FUNCTION_BLOCK EmergencyReactor_2 (* CAT Function Block Type *)
  (* Standard: 61499-2 *)
  (* Version 0.0, 7/4/2026, Schneider Electric, template *)
  PACKAGE SE.Nereda;
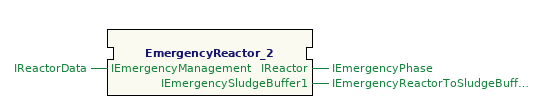
  SOCKETS
    IEmergencyManagement : IReactorData;
  END_SOCKETS
  PLUGS
    IReactor : IEmergencyPhase;
    IEmergencySludgeBuffer1 : IEmergencyReactorToSludgeBuffer;
  END_PLUGS
  (* 01 - FUNCTIONNAL INPUT INTERFACE *)
  (* 00 - INITIALIZATION *)
  (* 05 - LOGIC *)
  (* 06 - HMI INTERFACE *)
  (* 03 - FIELD INTERFACE *)
  (* 02 - FUNCTIONNAL OUTPUT INTERFACE *)
  (* Emergency Recipe Logic *)
  (* 04 - CHILDREN *)
  (* 4A - TYPICALS *)
  (* Reset Force Trs *)
  (* Skip Sludge Discharge Logic *)
  (* Steps Durations *)
  FBS
    INIT : plcStart(Prio := 50, Delay := T#0ms);
    IThis : EmergencyReactor_2_HMI(QI := TRUE);
    Step1_Feed : E_DELAY_V_D_ZERO;
    Step2_VentSludge : E_DELAY_V_D_ZERO;
    Step3_SludgeDischarge : E_DELAY_V_D_ZERO;
    Step4_LowerLevel : E_DELAY_V_D_ZERO;
    Step6_VentAerate : E_DELAY_V_D_ZERO;
    Step7_Wait : E_DELAY_V_D_ZERO;
    Step8_VentSludge : E_DELAY_V_D_ZERO;
    ResetTrsDelay : E_DELAY(DT := T#300ms);
    ResetTrs : TriggerNot0; {SET_ATTRIBUTE(Configuration.Component.HideUnusedPorts, )}
    SkipSludgeDischargeLogic : S1SkipS2(pin_EE0DFC875BC8FD2C := 3, pin_8745D113BFC82E09 := 9);
    SmoothSkip : boolValueChanged;
    EmergencyInitialisation : EmergencyInit2(pin_F6BF5230E0E343F0 := T#15m);
    S5_AerateTime : S5_AerateTime2;
    Step5_Aerate : COUNTER(pin_12B31DD3EC852BD8 := TRUE); {SET_ATTRIBUTE(Configuration.Component.HideUnusedPorts, )}
    ForceStopAeration : StopAerate2;
    FeedStarted : boolValueChanged;
    GoToS8 : OR_88A3DD8EC65DD11C; {SET_ATTRIBUTE(Configuration.GenericFBType.InterfaceParams, Runtime.Standard#CNT:=2;OUT:BOOL)}
    GoToS8Smooth : boolValueChanged;
    EmergencyRecipeSequence : EmergencyRecipeSequence_2;
    Step9_SludgeDischarge : E_DELAY_V_D_ZERO;
    Step10_Wait : E_DELAY_V_D_ZERO;
    Step6_VentAerate1 : E_DELAY_V_D_ZERO;
  END_FBS
  EVENT_CONNECTIONS
    IReactor.3CBA18632C5993F7 TO EmergencyRecipeSequence.5F230DB7635D55AE;
    IReactor.B9A3DD1A626C862D TO EmergencyRecipeSequence.5F230DB7635D55AE;
    IReactor.4DCB92F6993C5EE1 TO EmergencyRecipeSequence.5F230DB7635D55AE;
    IReactor.CF95EBECB4A2EBBE TO EmergencyRecipeSequence.5F230DB7635D55AE;
    IReactor.3F1D0A688A5176FD TO EmergencyRecipeSequence.5F230DB7635D55AE;
    IReactor.B334EFD88038E789 TO EmergencyRecipeSequence.5F230DB7635D55AE;
    Step1_Feed.1457E63E0C241C83 TO EmergencyRecipeSequence.62A0C79B5D89C4FB;
    Step2_VentSludge.1457E63E0C241C83 TO EmergencyRecipeSequence.24741A0901B103DB;
    Step3_SludgeDischarge.1457E63E0C241C83 TO EmergencyRecipeSequence.FEA4481ED0C2A43C;
    Step4_LowerLevel.1457E63E0C241C83 TO EmergencyRecipeSequence.9041C273A86FC2E4;
    Step6_VentAerate.1457E63E0C241C83 TO EmergencyRecipeSequence.5D1CA06DD981DC88;
    Step7_Wait.1457E63E0C241C83 TO EmergencyRecipeSequence.87133753EE03EF50;
    Step8_VentSludge.1457E63E0C241C83 TO EmergencyRecipeSequence.45085FB160311A79;
    SmoothSkip.CHD TO EmergencyRecipeSequence.3824F5F239920D6C;
    IReactor.1F4F3B9CDE5DCB1C TO EmergencyRecipeSequence.F6AE117EB4EE709F;
    IReactor.0001D958FDF5E959 TO EmergencyRecipeSequence.C960811A6435E9DC;
    EmergencyRecipeSequence.3B7FC9F46DCC7431 TO IReactor.42529785B6820948;
    EmergencyRecipeSequence.3B7FC9F46DCC7431 TO IReactor.B633B7A44F850807;
    EmergencyRecipeSequence.3B7FC9F46DCC7431 TO IReactor.B3BCF5E9C62C69B8;
    EmergencyRecipeSequence.3B7FC9F46DCC7431 TO IReactor.2000F66036015D52;
    EmergencyRecipeSequence.3B7FC9F46DCC7431 TO IReactor.8A3A142CC73C9F25;
    EmergencyRecipeSequence.BFFB06EAE80CA24C TO Step1_Feed.START;
    EmergencyRecipeSequence.899C844BE45E6C4D TO Step1_Feed.STOP;
    EmergencyRecipeSequence.758107C20AA8F48B TO Step2_VentSludge.START;
    EmergencyRecipeSequence.18CD3557BE39D07B TO Step2_VentSludge.STOP;
    EmergencyRecipeSequence.77F2040F9E65C9AB TO Step3_SludgeDischarge.START;
    EmergencyRecipeSequence.728874E1FE8923C2 TO Step3_SludgeDischarge.STOP;
    EmergencyRecipeSequence.F0D24A0013391FCB TO Step4_LowerLevel.START;
    EmergencyRecipeSequence.DBC21B10FAB6B6D6 TO Step4_LowerLevel.STOP;
    EmergencyRecipeSequence.5F688AB98BE3DBA8 TO Step5_Aerate.START;
    EmergencyRecipeSequence.CFC9FFB1D070A85D TO Step5_Aerate.STOP;
    EmergencyRecipeSequence.D93FC42377801178 TO Step6_VentAerate.START;
    EmergencyRecipeSequence.94B7CB1BE3844802 TO Step6_VentAerate.STOP;
    EmergencyRecipeSequence.D6AAA325013931BD TO Step7_Wait.START;
    EmergencyRecipeSequence.66DEB21CDAAC07A1 TO Step7_Wait.STOP;
    EmergencyRecipeSequence.4C7C51E8F73DAAF0 TO Step8_VentSludge.START;
    EmergencyRecipeSequence.4F8F2BAA25498729 TO Step8_VentSludge.STOP;
    Step1_Feed.INITO TO Step2_VentSludge.INIT;
    Step2_VentSludge.INITO TO Step3_SludgeDischarge.INIT;
    Step3_SludgeDischarge.INITO TO Step4_LowerLevel.INIT;
    Step4_LowerLevel.INITO TO Step6_VentAerate1.INIT;
    Step6_VentAerate.INITO TO Step7_Wait.INIT;
    Step7_Wait.INITO TO Step8_VentSludge.INIT;
    ResetTrs.4D14044435EE07B0 TO ResetTrsDelay.START;
    SkipSludgeDischargeLogic.9D8BC655F08DCD6C TO SmoothSkip.REQ;
    EmergencyRecipeSequence.556D2F5B235B9790 TO SkipSludgeDischargeLogic.74AB0FAFF377F024;
    IEmergencyManagement.E1D373823D64ACA0 TO IReactor.0FA2667D36826F2B;
    Step5_Aerate.INITO TO EmergencyInitialisation.7772EF333A96DB94;
    EmergencyInitialisation.5BE6234FD14189DB TO INIT.ACK_FIRST;
    EmergencyInitialisation.87FEA01C25C77B1D TO EmergencyRecipeSequence.4E3261F33DF95CD1;
    IEmergencyManagement.9D1E5F7369C5538B TO EmergencyInitialisation.E815AC1CDB9AD32A;
    IEmergencyManagement.E1D373823D64ACA0 TO EmergencyInitialisation.1FA17325B39B02F6;
    IEmergencyManagement.61CD32E3E6AEDF7D TO EmergencyInitialisation.5DED6604D26A7975;
    IEmergencyManagement.198EF041C70827BC TO S5_AerateTime.0D2EA60FD6C23367;
    IEmergencyManagement.1C1DD8946F24CFF9 TO S5_AerateTime.C7A276F0816E041D;
    S5_AerateTime.8B394E005AFEAD78 TO IEmergencyManagement.D499D06F1953A020;
    S5_AerateTime.8B394E005AFEAD78 TO Step5_Aerate.E9D3BB8F75D35902;
    IEmergencyManagement.7D5F3067068DE334 TO EmergencyRecipeSequence.25F0D728C2D36669;
    IEmergencyManagement.7D5F3067068DE334 TO IReactor.3CAF22C03BECB249;
    ForceStopAeration.7530111629E0F796 TO EmergencyRecipeSequence.56BBB9AD7704F212;
    IReactor.B9A3DD1A626C862D TO ForceStopAeration.D950482A44AC5C73;
    IEmergencyManagement.B3BDDBF095B97A2B TO ForceStopAeration.D950482A44AC5C73;
    IEmergencyManagement.E1D373823D64ACA0 TO EmergencyRecipeSequence.68E2F3B4BFF358D6;
    IReactor.3CBA18632C5993F7 TO FeedStarted.REQ;
    FeedStarted.CHD TO IEmergencyManagement.138EEC247A2C05E7;
    SkipSludgeDischargeLogic.5213FB99EC5BE951 TO ForceStopAeration.D950482A44AC5C73;
    EmergencyInitialisation.5BE6234FD14189DB TO EmergencyRecipeSequence.68E2F3B4BFF358D6;
    IEmergencyManagement.395F2A7D1AB6A478 TO EmergencyInitialisation.8D22CD40FC41E8B5;
    IEmergencyManagement.395F2A7D1AB6A478 TO EmergencyRecipeSequence.8BD9ED85505D599F;
    Step6_VentAerate1.INITO TO Step6_VentAerate.INIT;
    IEmergencyManagement.CF316F4BA7C11A07 TO EmergencyInitialisation.2B59ADD28234FD73;
    IEmergencyManagement.77175193A5DFB16A TO EmergencyRecipeSequence.CF595DA908C4D604;
    EmergencyRecipeSequence.556D2F5B235B9790 TO IEmergencyManagement.48081868B719DABE;
    IReactor.4DCB92F6993C5EE1 TO IEmergencyManagement.48081868B719DABE;
    GoToS8.CNF TO GoToS8Smooth.REQ;
    GoToS8Smooth.CHD TO EmergencyRecipeSequence.4E3261F33DF95CD1;
    EmergencyInitialisation.87FEA01C25C77B1D TO GoToS8.REQ;
    IEmergencyManagement.61CD32E3E6AEDF7D TO GoToS8.REQ;
    Step9_SludgeDischarge.INITO TO Step10_Wait.INIT;
    Step8_VentSludge.INITO TO Step9_SludgeDischarge.INIT;
    EmergencyRecipeSequence.159DAAF64474114A TO Step9_SludgeDischarge.START;
    EmergencyRecipeSequence.043FC99FF466ACE5 TO Step9_SludgeDischarge.STOP;
    EmergencyRecipeSequence.6D74F5F87D5293B0 TO Step10_Wait.START;
    EmergencyRecipeSequence.C125C1F9A17D8460 TO Step10_Wait.STOP;
    Step9_SludgeDischarge.1457E63E0C241C83 TO EmergencyRecipeSequence.CBB132F8E1E06425;
    Step10_Wait.1457E63E0C241C83 TO EmergencyRecipeSequence.2C1A1FFEA773D0E8;
    EmergencyRecipeSequence.3B7FC9F46DCC7431 TO IReactor.0F544A40694CE400;
    EmergencyRecipeSequence.556D2F5B235B9790 TO IReactor.DAE1720DE74FAACB;
    IEmergencyManagement.93812D9FEC4294F9 TO EmergencyRecipeSequence.035DD9202D5272B8;
    Step10_Wait.INITO TO Step5_Aerate.INIT;
    EmergencyRecipeSequence.5F688AB98BE3DBA8 TO Step6_VentAerate1.START;
    EmergencyRecipeSequence.CFC9FFB1D070A85D TO Step6_VentAerate1.STOP;
    Step6_VentAerate1.1457E63E0C241C83 TO EmergencyRecipeSequence.AA8C7EBD4EBD70F0;
    IReactor.2DDA8AB533D7441D TO EmergencyRecipeSequence.1E0B2A3AB6A90076;
    IEmergencyManagement.E1D373823D64ACA0 TO IEmergencySludgeBuffer1.D46CB75BB047204F;
    IReactor.3CBA18632C5993F7 TO IEmergencySludgeBuffer1.3F9F1A3D0BC5ACBF;
    IEmergencyManagement.7D5F3067068DE334 TO IEmergencySludgeBuffer1.69A30D6F1EEC778E;
    INIT.FIRST_INIT TO IThis.11B0EEC0AF1F6F5A;
    INIT.REDO_INIT TO IThis.11B0EEC0AF1F6F5A;
    EmergencyRecipeSequence.556D2F5B235B9790 TO IThis.C39B00E2AD0232CC;
    IEmergencyManagement.E1D373823D64ACA0 TO IThis.C454C4B6A808EB9F;
    ResetTrsDelay.EO TO IThis.908B60AA8FD99187;
    IThis.7797C5138BE465AE TO IThis.D73F4F826029EE6B;
    S5_AerateTime.8B394E005AFEAD78 TO IThis.188CF7222009AE29;
    ForceStopAeration.5ED5F3C70645AC06 TO IThis.188CF7222009AE29;
    S5_AerateTime.878A4998A65F56E0 TO IThis.7360449561F94EA9;
    Step5_Aerate.INITO TO IThis.9D2FDC03CB586F4F;
    IEmergencyManagement.7D5F3067068DE334 TO IThis.FD84EE6824F2A446;
    IThis.69E91E9E46EEE4A5 TO Step1_Feed.INIT;
    IThis.7C2D7DF8D7E29126 TO ResetTrs.98B4D14610C64DF9;
    IThis.7C2D7DF8D7E29126 TO EmergencyRecipeSequence.56F42E6AA601D269;
    IThis.A02D1390759D9486 TO EmergencyInitialisation.4A8FE6F9318E2B02;
    IThis.A02D1390759D9486 TO S5_AerateTime.0D2EA60FD6C23367;
    IThis.A02D1390759D9486 TO ForceStopAeration.D950482A44AC5C73;
    IThis.1D92FE3FE5B995E2 TO IReactor.BC34E8F0E0F52444;
    IThis.621A8557BCE5A33F TO IReactor.1BDE0720AC8B4391;
    IThis.72CBF4E7BB40B16D TO IReactor.FF8E2C9D67AADBF4;
    IThis.024A635046F06C0B TO IReactor.4E395DC016F294D9;
  END_CONNECTIONS
  DATA_CONNECTIONS
    EmergencyRecipeSequence.8B42F21C51560908 TO IReactor.8B7B31E6EA54014D;
    EmergencyRecipeSequence.A11B93FCF2C8455F TO IReactor.09084E8C7BADBD46;
    EmergencyRecipeSequence.2A15B42D80F87BCA TO IReactor.C947D1396F3B0873;
    EmergencyRecipeSequence.EC54CA5500C858C1 TO IReactor.419E697BA1D2FB08;
    EmergencyRecipeSequence.A9E8FE003DEE6E89 TO IReactor.C584AEAB998AB515;
    IReactor.599667ECF678E518 TO EmergencyRecipeSequence.02C5FE17473E63ED;
    IReactor.656FC0E59D395E4C TO EmergencyRecipeSequence.9F29B8C1612DCC07;
    IReactor.9CFBB312DE29B9C4 TO EmergencyRecipeSequence.ED57F4FA4B77207F;
    IReactor.A1460632301E8B7F TO EmergencyRecipeSequence.89F466D1EDD34A8F;
    IReactor.A92252B4F4DF917A TO EmergencyRecipeSequence.5FBA38ABF9198C98;
    Step1_Feed.716D3F3042596C89 TO EmergencyRecipeSequence.CA116731A496187E;
    Step2_VentSludge.716D3F3042596C89 TO EmergencyRecipeSequence.356882B50FEB9A7D;
    Step3_SludgeDischarge.716D3F3042596C89 TO EmergencyRecipeSequence.111361C8BEDF440B;
    Step4_LowerLevel.716D3F3042596C89 TO EmergencyRecipeSequence.82CEB92F735FC5D4;
    Step6_VentAerate.716D3F3042596C89 TO EmergencyRecipeSequence.0228D93DF2A0E691;
    Step7_Wait.716D3F3042596C89 TO EmergencyRecipeSequence.F00C171ABB730806;
    Step8_VentSludge.716D3F3042596C89 TO EmergencyRecipeSequence.0EEA3AF033FFC1FD;
    SmoothSkip.Output TO EmergencyRecipeSequence.43A591812296CA90;
    IReactor.579DEB3758BDB938 TO EmergencyRecipeSequence.7A1CAB8AE52AE374;
    IReactor.1156E288C0C38120 TO EmergencyRecipeSequence.CB5D14E9C5586FB9;
    SkipSludgeDischargeLogic.DBD9C05F71A70F66 TO SmoothSkip.Input;
    EmergencyRecipeSequence.1A64065878672AC0 TO SkipSludgeDischargeLogic.2058267BFC81675C;
    IEmergencyManagement.F0BEEA13B7FB6780 TO IReactor.5159724764416574;
    EmergencyInitialisation.AC3533DBCBFC24D5 TO EmergencyRecipeSequence.73A0EB798F8AE64D;
    GoToS8Smooth.Output TO EmergencyRecipeSequence.8C498327642AF905;
    IEmergencyManagement.7614E537E01F969F TO EmergencyInitialisation.C2EDD382E854309C;
    IEmergencyManagement.852A82A24B95110C TO EmergencyInitialisation.8DFF8A8B75E55DBC;
    IEmergencyManagement.F0BEEA13B7FB6780 TO EmergencyInitialisation.5CEC0909DD41DD44;
    IEmergencyManagement.074948F0B024FF2E TO EmergencyInitialisation.417A4B99C6EAD037;
    IEmergencyManagement.758E7E3A994DF6A3 TO S5_AerateTime.051E4CDC84405E95;
    IEmergencyManagement.90388C221FF11A3D TO S5_AerateTime.4E488DE24686A5F2;
    S5_AerateTime.3E8F4A267A25DD05 TO IEmergencyManagement.793E1D04BE895F4E;
    S5_AerateTime.6A9E00F95DC3CAB2 TO IEmergencyManagement.3807C75A82F33B22;
    S5_AerateTime.3E8F4A267A25DD05 TO Step5_Aerate.2BD9889911508ED1;
    IEmergencyManagement.35F3027F47B7A966 TO EmergencyRecipeSequence.53ADC5A2738A60DC;
    IEmergencyManagement.35F3027F47B7A966 TO IReactor.63583CB69DED3592;
    ForceStopAeration.8A55773E02AECBCB TO EmergencyRecipeSequence.F39141D7A6A53184;
    IReactor.A63167A113600EB8 TO ForceStopAeration.19D48581CC6CEC95;
    IEmergencyManagement.83DE9B371B83EBB9 TO ForceStopAeration.20B8DEE9B9067A7E;
    IEmergencyManagement.F0BEEA13B7FB6780 TO EmergencyRecipeSequence.C537A25E1616B854;
    IReactor.F208B10244BCFEF2 TO FeedStarted.Input;
    FeedStarted.Output TO IEmergencyManagement.1D99A7E687AA4E06;
    IEmergencyManagement.3C27B3AC98B413B4 TO EmergencyInitialisation.79C2DD791585EF12;
    SkipSludgeDischargeLogic.59D0E2CFD06FCCA4 TO ForceStopAeration.E5E5D63C44355F3C;
    SkipSludgeDischargeLogic.BEF2F356EA04F63C TO ForceStopAeration.11917BAB3534074F;
    IEmergencyManagement.B1FC30AB336AE8E9 TO EmergencyRecipeSequence.EB24B639967D6395;
    EmergencyInitialisation.511C6D20E2A2A314 TO EmergencyRecipeSequence.A0CAD84FAFB4D508;
    IEmergencyManagement.B1FC30AB336AE8E9 TO EmergencyInitialisation.0058582DF67974BB;
    IEmergencyManagement.7FC77B7D4B4A5A4D TO EmergencyInitialisation.E3C04CDD1BC5A85D;
    IEmergencyManagement.B7D7393A43236C58 TO EmergencyInitialisation.9E91693CC077CF71;
    IEmergencyManagement.EEDAEC65A069032E TO EmergencyRecipeSequence.DB0738E6DF6AD68E;
    EmergencyRecipeSequence.1A64065878672AC0 TO IEmergencyManagement.613E286D19768818;
    IReactor.9CFBB312DE29B9C4 TO IEmergencyManagement.B3BCA5E1F4B3D013;
    GoToS8.OUT TO GoToS8Smooth.Input;
    EmergencyInitialisation.DF25ED8EB3FED3D4 TO GoToS8.IN1;
    IEmergencyManagement.713BAA92BE7C280E TO GoToS8.IN2;
    EmergencyRecipeSequence.05803EDF26892491 TO IReactor.198FB8D9804ED082;
    EmergencyRecipeSequence.4076D29063AB0B00 TO IReactor.486306180C62B9EF;
    IReactor.E996774D431E1B79 TO EmergencyRecipeSequence.A2ED29C3A4B57D44;
    IReactor.800D089965342DF6 TO EmergencyRecipeSequence.69F1D0FE13048380;
    Step9_SludgeDischarge.716D3F3042596C89 TO EmergencyRecipeSequence.CC3E20D91936F86E;
    Step10_Wait.716D3F3042596C89 TO EmergencyRecipeSequence.34AB02FCEF6642EF;
    IEmergencyManagement.1675BB23EEFCF5E9 TO EmergencyRecipeSequence.5989C017FA1C720B;
    Step6_VentAerate1.716D3F3042596C89 TO EmergencyRecipeSequence.CC0CCEB2D046659B;
    IReactor.C54C3886CAD71D0C TO EmergencyRecipeSequence.ACB986D17AA81EAF;
    IEmergencyManagement.F0BEEA13B7FB6780 TO IEmergencySludgeBuffer1.128C534CB06CDD0F;
    IReactor.D62F1904A2304A82 TO IEmergencySludgeBuffer1.D455BE5F3243F8CD;
    IReactor.EDD981DC30DF57BC TO IEmergencySludgeBuffer1.98FFA78276DA0653;
    IReactor.DA119668EC2B3E62 TO IEmergencySludgeBuffer1.2680CB24DDCC2D3E;
    IEmergencyManagement.35F3027F47B7A966 TO IEmergencySludgeBuffer1.A351B45A56D7A52F;
    EmergencyRecipeSequence.1A64065878672AC0 TO IThis.B3535F417A0074C5;
    IEmergencyManagement.F0BEEA13B7FB6780 TO IThis.71DB4288F980DD7A;
    IThis.F0EDDD752FB146AF TO IThis.2A6B48A49CC51EE0;
    S5_AerateTime.3E8F4A267A25DD05 TO IThis.0DCF6DA005733527;
    ForceStopAeration.C8B85A94FE68EF0C TO IThis.71E3BF00CD92D001;
    S5_AerateTime.4CD884F27F8D62DD TO IThis.A4518E9C005FED53;
    IEmergencyManagement.35F3027F47B7A966 TO IThis.7498551BC2E13233;
    IThis.5C9558FA20CCCAFB TO ResetTrs.622EA78CA147C620;
    IThis.5C9558FA20CCCAFB TO EmergencyRecipeSequence.1EFAFB1416CAAE87;
    IThis.D3644ED70524C0F1 TO Step1_Feed.DT1;
    IThis.D3644ED70524C0F1 TO S5_AerateTime.C5F8AE19B1F00F21;
    IThis.33D4356E329ECCF2 TO Step2_VentSludge.DT1;
    IThis.33D4356E329ECCF2 TO S5_AerateTime.E8F6A7D9DCD9BBE1;
    IThis.9B01CEED6ECAE668 TO Step3_SludgeDischarge.DT1;
    IThis.9B01CEED6ECAE668 TO EmergencyInitialisation.948836585F0EEA5B;
    IThis.9B01CEED6ECAE668 TO S5_AerateTime.BBEC65C254C77C0B;
    IThis.11E3ABF20E7068A4 TO Step4_LowerLevel.DT1;
    IThis.11E3ABF20E7068A4 TO EmergencyInitialisation.0CD3D5D316F69EF0;
    IThis.11E3ABF20E7068A4 TO S5_AerateTime.987FE50D3182D670;
    IThis.B750E161B72BAAC1 TO Step6_VentAerate1.DT1;
    IThis.036FF5CCE7E00472 TO Step6_VentAerate.DT1;
    IThis.036FF5CCE7E00472 TO EmergencyInitialisation.167B000B6721BF5C;
    IThis.036FF5CCE7E00472 TO ForceStopAeration.02B77BABB54CA7BE;
    IThis.036FF5CCE7E00472 TO S5_AerateTime.03FA70645F2696D4;
    IThis.C90D68E8BE4DBE36 TO ForceStopAeration.E68AB0318ABA2B14;
    IThis.C90D68E8BE4DBE36 TO Step7_Wait.DT1;
    IThis.C90D68E8BE4DBE36 TO EmergencyInitialisation.CFBCABADFC8098AD;
    IThis.C90D68E8BE4DBE36 TO S5_AerateTime.F499F59EB03E2123;
    IThis.C25432226AC2046D TO Step8_VentSludge.DT1;
    IThis.C25432226AC2046D TO EmergencyInitialisation.38D26424A39E04A0;
    IThis.C25432226AC2046D TO S5_AerateTime.F9726491C55C37B7;
    IThis.C3D0734543022201 TO S5_AerateTime.0730E12942861AFC;
    IThis.C3D0734543022201 TO Step9_SludgeDischarge.DT1;
    IThis.C3D0734543022201 TO EmergencyInitialisation.E4383207F02C387C;
    IThis.AEBBF7743AEFCC72 TO Step10_Wait.DT1;
    IThis.AEBBF7743AEFCC72 TO EmergencyInitialisation.AAD116E9F3FCBC75;
    IThis.AEBBF7743AEFCC72 TO S5_AerateTime.9ED54AAE61E0A080;
    IThis.22F6EB8128B0DB9A TO IReactor.34423AC7BCF3714C;
    IThis.E80EF6313E2D5B22 TO IReactor.8B46E1E2CAE6076D;
    IThis.AB1D55433D4D5D68 TO IReactor.A29A102F17AA7B5F;
    IThis.3B07507DE970AEED TO IReactor.EC5E58B468310216;
    IThis.E8500FD902693DE1 TO IReactor.51705890CC419D73;
    IThis.B9A6F8131C758152 TO IReactor.F44F737D6F09989F;
    IThis.FBAC05C2DEE3E62F TO IReactor.86DD4C5333164B26;
    IThis.C25432226AC2046D TO ForceStopAeration.5E61F739B3DD3A6C;
    IThis.C3D0734543022201 TO ForceStopAeration.67A808A4C7D6712E;
    IThis.AEBBF7743AEFCC72 TO ForceStopAeration.9CD228C4598ACEF5;
  END_CONNECTIONS
END_FUNCTION_BLOCK
